PROGRAM PhotoLumBkgrdSerialCom
VAR_INPUT
	Config : PhotoLumConfig;
END_VAR
VAR
END_VAR

// AxisConfigs
IF Config.AxesConfigs.Ps10OwisAxisConfig.IsEnabled THEN
	BkgrdSerialOwisPs10();	
END_IF

// LightConfigs
IF Config.LightConfigs.ArduinoLightConfig.IsEnabled THEN
	BkgrdSerialLight();
ELSIF Config.LightConfigs.EvosensLightConfig.IsEnabled THEN
	BkgrdSerialLight();
END_IF

END_PROGRAM

(* stored: Version 1.1.0.1, ProductVersion 3.1.4024.12
   POU PhotoLumBkgrdSerialCom: Id {60e560e3-a6b9-4afb-851a-68818bf21bef}, SpecialFunc None *)
